TYPE ST_MachineMode :
STRUCT
	/// Operation Mode 
	Standby: BOOL;
	Manual: BOOL;
	MDI: BOOL;
	Automatic: BOOL;
	///REFERENCE		: BOOL;  TC3HR
	Homing: BOOL;
	/// Operation State
	Select : BOOL; 
	Ready  : BOOL;
	Start: BOOL;
	Stop: BOOL;
	Reset: BOOL;
	Error: BOOL;
	/// Special functions 
	ChannelSignals: ST_ChannelSignals;
	BlockSearch: ST_BlockSearch;
	SyntaxCheck: ST_SyntaxCheck;
	ManualMode: ST_ManualMode;
	/// Strings 
	ProgramName: STRING(1024);
	MDIString: STRING(1024);
END_STRUCT
END_TYPE

(* stored: Version 1.1.0.1, ProductVersion 3.1.4022.6
   DUT ST_MachineMode: Id {bedbe333-fa74-44a4-9ca4-ab8d537f835e} *)
